{attribute 'qualified_only'}
VAR_GLOBAL
	
	// binary inputs
	//biPowerFault				AT %I* : BOOL;
	biTankFloodFault			AT %I* : BOOL;
	biLS1_WaterMidLevel			AT %I* : BOOL;
	biLS2_WaterHighLevel		AT %I* : BOOL;
	biLS3_WaterLowLevel			AT %I* : BOOL;
	//biPS1_						AT %I* : BOOL;
	                        	
	// binary outputs       	
	boSV1_DrainValve			AT %Q* : BOOL;
	boSV2_SpaValve				AT %Q* : BOOL;
	boSV3_DeliveryValve			AT %Q* : BOOL;
	boSV4_WaterInletValve		AT %Q* : BOOL;
	boH1_UpstreamHeater			AT %Q* : BOOL;
	boH2_SpaHeater				AT %Q* : BOOL;
	boH3_FlowmeterHeater		AT %Q* : BOOL;
	boH4_ExternalHeater			AT %Q* : BOOL;
	//boLED1_ReadyLight			AT %Q* : BOOL;
	//boLED2_AlarmLight			AT %Q* : BOOL;
	
	// analog inputs
	aiPT1_UpstreamPressure		AT %I* : INT;
	aiPT2_DownstreamPressure 	AT %I* : INT;
	aiTC1_SpaTemp				AT %I* : INT;
	aiTC2_FlometerTemp			AT %I* : INT;
	aiTC3_ExternalTemp			AT %I* : INT;
	aiTC4_DeliveryTemp			AT %I* : INT;	
	
END_VAR

(* stored: Version 1.1.0.1, ProductVersion 3.1.4026.19
   GVL GVL_IO: Id {2a04d97b-78dd-4508-9070-7a711c04c75b} *)
